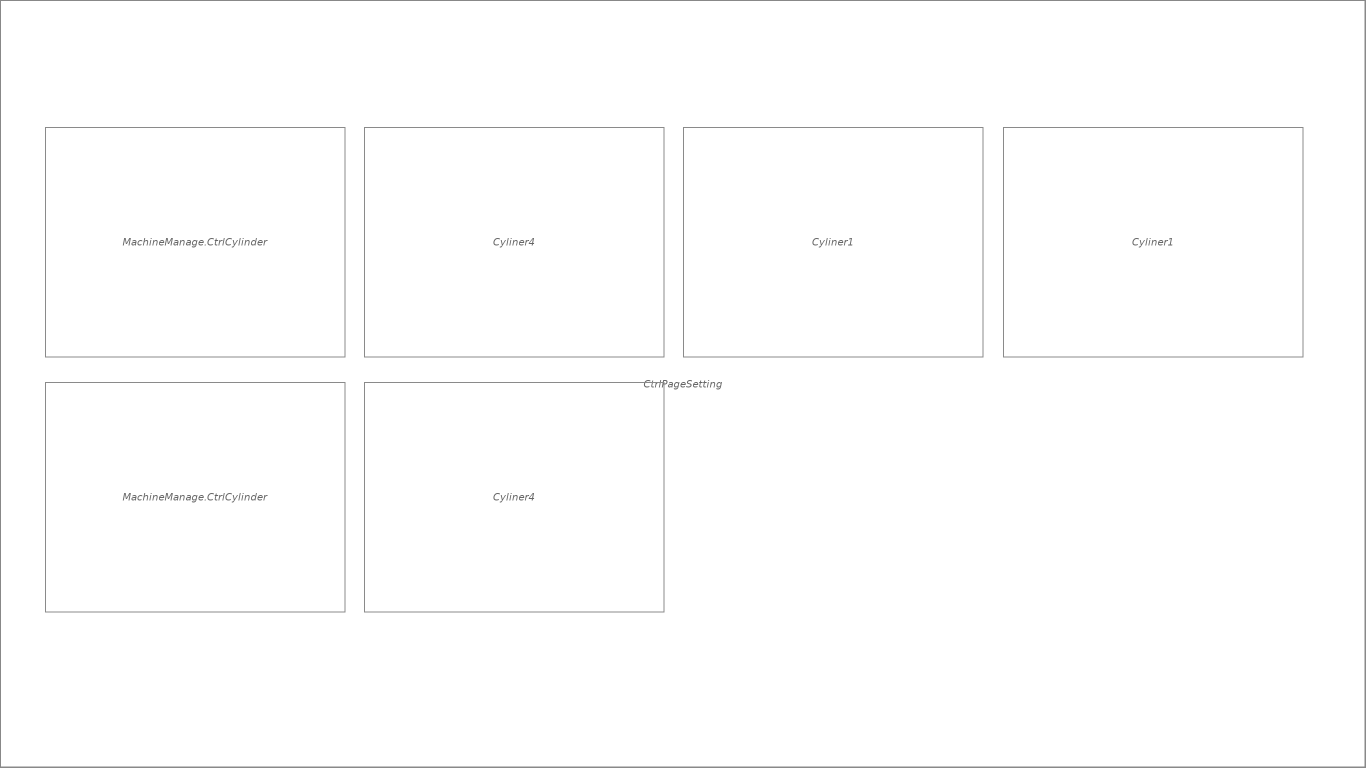
VISUALIZATION PageSetting_Unload_L  // 1366x768
    Frame (0,0 1366x768)
        shows CtrlPageSetting()
    Frame (683,127 300x230)
        shows Cyliner1(System := G_stSystem, Cylinder := G_arrCylinder[E_Cylinder.UnloadUcBeltTipper], CylinderData := G_arrCylinderData[E_Cylinder.UnloadUcBeltTipper])
    Frame (1003,127 300x230)
        shows Cyliner1(System := G_stSystem, Cylinder := G_arrCylinder[E_Cylinder.UnloadUcBeltLift], CylinderData := G_arrCylinderData[E_Cylinder.UnloadUcBeltLift])
    Frame (45,127 300x230)
        shows MachineManage.CtrlCylinder(System := G_stSystem, Cylinder := G_arrCylinder[E_Cylinder.UnloadFrockConveyorPrevent], CylinderData := G_arrCylinderData[E_Cylinder.UnloadFrockConveyorPrevent])
    Frame (364,127 300x230)
        shows Cyliner4(System := G_stSystem, Cylinder := G_arrCylinder[E_Cylinder.UnloadFrockConveyorPush], CylinderData := G_arrCylinderData[E_Cylinder.UnloadFrockConveyorPush])
    Frame (45,382 300x230)
        shows MachineManage.CtrlCylinder(System := G_stSystem, Cylinder := G_arrCylinder[E_Cylinder.UnloadUcElevator], CylinderData := G_arrCylinderData[E_Cylinder.UnloadUcElevator])
    Frame (364,382 300x230)
        shows Cyliner4(System := G_stSystem, Cylinder := G_arrCylinder[E_Cylinder.UnloadUcConveyorPush], CylinderData := G_arrCylinderData[E_Cylinder.UnloadUcConveyorPush])
END_VISUALIZATION

(* stored: Version 1.1.0.1, ProductVersion 3.1.4024.3
   Visu PageSetting_Unload_L: Id {38f26bb5-cf58-49ca-9b42-9bef9bb70420} *)
